FUNCTION_BLOCK EventLoggerClass IMPLEMENTS IEventLoggers
VAR_INPUT
END_VAR
VAR_OUTPUT
END_VAR
VAR
    fbMsg : FB_TcMessage; 
	fbTest : Tc3_EventLogger.FB_TcEvent;
	fbInfo : Tc3_EventLogger.FB_TcSourceInfo;
	LogLevel : TcEventSeverity;	
END_VAR

METHOD PUBLIC Send : BOOL
VAR_INPUT
	eventType : Tc3_EventLogger.TcEventEntry;
	args : STRING(255);
END_VAR
THIS^.fbMsg.CreateEx(eventType, 0);
THIS^.fbMsg.ipArguments.AddString(args);
THIS^.fbMsg.Send(0);
THIS^.fbMsg.Release();
END_METHOD

END_FUNCTION_BLOCK

(* stored: Version 1.1.0.1, ProductVersion 3.1.4024.11
   POU EventLoggerClass: Id {3f6e8d91-2b3f-4c47-b9e7-0101dde119b9}, SpecialFunc None
   Method Send: Id {ae7ec69f-155c-4e06-b3b3-42ff1592972e} *)
